PROGRAM B_4_2_PRG_Master_ProcessDoor

VAR

	bEventsFlag							: ARRAY [0..100] OF BOOL;
/////////////////////////////////////////////////////////////////////////////////////I O/////////////////////////////////////////////////////////////////////////////////////	
	
	bOpenDoor							: BOOL;
	bCloseDoor							: BOOL;
	bDoorClosed							: BOOL;
	bDoorOpened							: BOOL;
	tonDoorOpened						: TON;

	
END_VAR

d_ACT_Set_Events_Station_4B();
a_ACT_Ctrl_Station_4B();
b_ACT_IO_B();
c_Manual();

ACTION a_ACT_Ctrl_Station_4B:
/////////////////////////////////////////////////////////////////////////////////////UTILITIES/////////////////////////////////////////////////////////////////////////////////////

/////////////////////////////////////////////////////////////////////////////////////CONDITIONS/////////////////////////////////////////////////////////////////////////////////////
IF stProcessDoor.CMD.bAbort THEN
	
	stProcessDoor.State				:= E_ProcessDoor_State.RESET;
	
ELSIF stProcessDoor.CMD.bEndCycle THEN
	
	stProcessDoor.State				:= E_ProcessDoor_State.STOPPING;

END_IF

CASE stProcessDoor.State OF
	
	E_ProcessDoor_State.ABORTED:
	
								IF stProcessDoor.CMD.bEnable THEN
									
									stProcessDoor.State				:= E_ProcessDoor_State.READY;
								
								END_IF
	
	E_ProcessDoor_State.READY:
	
								IF stProcessDoor.CMD.bExecute AND 	stProcessDoor.CMD.ProcessDoorCMD.OpenDoor	THEN

									stProcessDoor.State				:= E_ProcessDoor_State.OPEN;
									
								ELSIF stProcessDoor.CMD.bExecute AND 	stProcessDoor.CMD.ProcessDoorCMD.CloseDoor	THEN
									
									stProcessDoor.State				:= E_ProcessDoor_State.CLOSE;									
																		
								END_IF
	
	E_ProcessDoor_State.OPEN:
	
								bOpenDoor							:= TRUE;
								
								IF bDoorOpened	THEN
									
									stProcessDoor.State				:= E_ProcessDoor_State.DONE;
								
								END_IF
								
	E_ProcessDoor_State.CLOSE:
	
								bCloseDoor							:= TRUE;
								
								IF bDoorClosed THEN
									
									stProcessDoor.State				:= E_ProcessDoor_State.DONE;
								
								END_IF
								
	E_ProcessDoor_State.DONE:
	
								bOpenDoor							:= FALSE;
								bCloseDoor							:= FALSE;
	
								IF stProcessDoor.CMD.bAcknowledge THEN
									
									stProcessDoor.CMD.bAcknowledge	:= FALSE;
									stProcessDoor.State				:= E_ProcessDoor_State.RESET;
								
								END_IF
	
	
	E_ProcessDoor_State.RESET:	
	
								bOpenDoor							:= FALSE;
								bCloseDoor							:= FALSE;
								
								IF NOT stProcessDoor.CMD.bAbort AND NOT stProcessDoor.CMD.bEndCycle THEN
									
									stProcessDoor.State				:= E_ProcessDoor_State.OPEN;
									
								ELSE stProcessDoor.State			:= E_ProcessDoor_State.ABORTED;
								END_IF
	
					
	E_ProcessDoor_State.STOPPING:					
									
								bOpenDoor							:= TRUE;
									
								IF bDoorOpened THEN
									
									bOpenDoor						:= FALSE;
									stProcessDoor.State				:= E_ProcessDoor_State.RESET;
								
								END_IF
								
							
														
									

ELSE stProcessDoor.State		:= E_ProcessDoor_State.ABORTED;
	
END_CASE
/////////////////////////////////////////////////////////////////////////////////////STATUS/////////////////////////////////////////////////////////////////////////////////////

stProcessDoor.Status.bBusy			:= 	stProcessDoor.State	= E_ProcessDoor_State.CLOSE OR
										stProcessDoor.State	= E_ProcessDoor_State.OPEN;
								
stProcessDoor.Status.bDone			:=	stProcessDoor.State	= E_ProcessDoor_State.DONE;

stProcessDoor.Status.bReady			:= 	stProcessDoor.State	= E_ProcessDoor_State.READY;

stProcessDoor.Status.bStopped		:= 	NOT stProcessDoor.Status.bBusy;
END_ACTION

ACTION b_ACT_IO_B:
tonDoorOpened( IN := NOT bDoorClosed AND bDoorOpeningFlag	, PT := stTimers.tDoorOpenedSignal);


bDoorClosed								:= dw_T05_EL1918.iProcessDoorClosed1 AND dw_T05_EL1918.iProcessDoorClosed2 AND dw_T05_EL1918.iProcessDoorFB;
bDoorOpened								:= tonDoorOpened.Q; 

dw_T09_EL2809.qOpenProcessDoor	:= bOpenDoor OR bProcessDoor_Up;	
dw_T09_EL2809.qCloseProcessDoor	:= bCloseDoor OR bProcessDoor_Down;
END_ACTION

ACTION c_Manual:
IF bProcessDoor_Up THEN
	
	bOpenDoor						:= TRUE;
	
ELSIF bDoorOpened THEN
	
	bOpenDoor						:= FALSE;

END_IF

IF  bProcessDoor_Down THEN
	
	bCloseDoor						:= TRUE;
	
ELSIF bDoorClosed THEN
	
	bCloseDoor						:= FALSE;

END_IF
END_ACTION

ACTION d_ACT_Set_Events_Station_4B:
//IMMEDIATE FAULTS

stStationEvents[4].aEvents[0].bEventTimer( IN := bCloseDoor AND NOT bDoorClosed, PT := T#5S);
stStationEvents[4].aEvents[0].bFault						:= TRUE;
stStationEvents[4].aEvents[0].bEventFlag					:= stStationEvents[4].aEvents[0].bEventTimer.Q;
stStationEvents[4].aEvents[0].bEventText					:= 'Process Door extend timeout';
stStationEvents[4].aEvents[0].sSolution						:= 'Check cylinders, neumatic connections and sensors';



//CYCLE STOP REQUEST

(*stStationEvents[4].aEvents[2].bCycleStopRequest			:= TRUE;
stStationEvents[4].aEvents[2].bEventFlag					:= bEventsFlag[2];
stStationEvents[4].aEvents[2].bEventText					:= 'ST1 EVENT 7';*)
END_ACTION

END_PROGRAM

(* stored: Version 1.1.0.1, ProductVersion 3.1.4026.17
   POU B_4_2_PRG_Master_ProcessDoor: Id {53a11cee-2388-4375-a004-26a2c48b086a}, SpecialFunc None
   Action a_ACT_Ctrl_Station_4B: Id {08b1d871-01b9-45fa-bb18-30d558502fc6}
   Action b_ACT_IO_B: Id {7a24ac88-21cc-4219-af73-2aba76419ebf}
   Action c_Manual: Id {af74f668-26ed-493a-861d-9af0f131bf72}
   Action d_ACT_Set_Events_Station_4B: Id {6917e64e-8f14-430a-8afe-2820b830fd4d} *)
